(* CODESYS project tcprocess.library
   Company: TcNexa
   DefaultNamespace: TcNexa_Components_TcProcess
   Version: 1.0.0.0
   Placeholder: TcProcess
   Author: ATI Software Engineering
   Description: This library serves as a valuable resource for managing reusable components within your automation projects
   Title: TcProcess

Project tree, tasks and I/O mapping:
  libraries: Tc2_Standard, * (Beckhoff Automation GmbH); Tc2_System, * (Beckhoff Automation GmbH); Tc3_Module, * (Beckhoff Automation GmbH); TcUnit, * (www.tcunit.org)
  Process Method Response/
    function block FB_MethodResponse [ST]: _clear, busy, description, error, copyFrom, setBusy, setFail, setPass
    function block FB_MethodResponse_1 [ST]: _clear, _formatDescription, _formatErrorMsg, busy, description, error, errorId, errorMsg, errorSrc, statusId, statusMsg, copyFrom, setBusy, setFail, setPass
  Process Step/
    function block FB_ProcessStep [ST]: actual, FB_main, inc, init, onEntry, onExit, set
  Tests/
    function block FB_MethodResponse_Test [ST]: _t_01_SetResponsePass_ExpectResponsePass, _t_02_SetResponseFail_ExpectResponseFail, _t_03_SetResponseBusy_ExpectResponseBusy, _t_04_CopyFrom_ExpectSameResponse
    function block FB_ProcessStep_Test [ST]: _t_01_StepInc_ExpectStepInc, _t_02_StepSet100_ExpectStep100, _t_03_StepManagment
    program PRG_TEST [ST]
  Version/
    global variables Global_Version
*)

// Version/Global_Version
{attribute 'TcGenerated'}
{attribute 'no-analysis'}
{attribute 'linkalways'}
// This function has been automatically generated from the project information.
VAR_GLOBAL CONSTANT
	{attribute 'const_non_replaced'}
	stLibVersion_TcProcess : ST_LibVersion := (iMajor := 1, iMinor := 0, iBuild := 0, iRevision := 0, nFlags := 0, sVersion := '1.0.0.0');
END_VAR

// Process Method Response/FB_MethodResponse
FUNCTION_BLOCK FB_MethodResponse
VAR
	_busy			: BOOL;						// Indicates if the method call is in progress
	_error			: BOOL;						// Indicates if the method call failed
	_description	: Tc2_System.T_MaxString;	// Information to show to the user
	
	
	
	
//	_statusMsg		: Tc2_System.T_MaxString;	// Status message from method call
//	_statusId		: UDINT;					// Message ID from method call, for further processing (translation etc.)
//	_errorMsg		: Tc2_System.T_MaxString;	// Error message from method call
//	_errorId		: UDINT;					// Error ID from method call
//	_errorSrc		: STRING;					// Source for the error (Beckhoff, Keyence etc.)
END_VAR

METHOD PROTECTED _clear
VAR_INPUT
END_VAR
_busy:= FALSE;
_error:= FALSE;
_description:= '';
END_METHOD

PROPERTY PUBLIC busy : BOOL
GET
busy:= _busy;
END_GET
END_PROPERTY

PROPERTY PUBLIC description : Tc2_System.T_MaxString
GET
description:= _description;
END_GET
END_PROPERTY

PROPERTY PUBLIC error : BOOL
GET
error:= _error;
END_GET
END_PROPERTY

METHOD PUBLIC copyFrom
VAR_INPUT
	Response		: FB_MethodResponse;
END_VAR
_busy:= Response.busy;
_error:= Response.error;
_description:= Response.description;
END_METHOD

METHOD PUBLIC setBusy
VAR_INPUT
	description	 	: Tc2_System.T_MaxString;
END_VAR
_clear();

_busy:= TRUE;
_description:= description;
END_METHOD

METHOD PUBLIC setFail
VAR_INPUT
	description	 	: Tc2_System.T_MaxString;
END_VAR
_clear();

_error:= TRUE;
_description:= description;
END_METHOD

METHOD PUBLIC setPass
VAR_INPUT
END_VAR
_clear();
END_METHOD

END_FUNCTION_BLOCK

// Process Method Response/FB_MethodResponse_1
FUNCTION_BLOCK FB_MethodResponse_1
VAR
	_busy			: BOOL;						// Indicates if the method call is in progress
	_error			: BOOL;						// Indicates if the method call failed
	_description	: Tc2_System.T_MaxString;	// Status and error message combined from method call
	_statusMsg		: Tc2_System.T_MaxString;	// Status message from method call
	_statusId		: UDINT;					// Message ID from method call, for further processing (translation etc.)
	_errorMsg		: Tc2_System.T_MaxString;	// Error message from method call
	_errorId		: UDINT;					// Error ID from method call
	_errorSrc		: STRING;					// Source for the error (Beckhoff, Keyence etc.)
END_VAR

METHOD PROTECTED _clear
VAR_INPUT
END_VAR
_busy:= FALSE;
_error:= FALSE;
_description:= '';
_statusMsg:= '';
_statusId:= 0;
_errorMsg:= '';
_errorId:= 0;
_errorSrc:= '';
END_METHOD

METHOD PROTECTED _formatDescription
VAR_INPUT
END_VAR
IF (_statusMsg <> '') AND (_errorMsg <> '') THEN
	_description:= Tc2_Standard.CONCAT(
		STR1:= _statusMsg,
		STR2:= ' -> ');
	_description:= Tc2_Standard.CONCAT(
		STR1:= _description,
		STR2:= _errorMsg);
ELSIF (_statusMsg <> '') THEN
	_description:= _statusMsg;
ELSIF (_errorMsg <> '') THEN
	_description:= _errorMsg;
END_IF
END_METHOD

METHOD PROTECTED _formatErrorMsg
VAR_INPUT
	
END_VAR
IF (_errorMsg = '') THEN
	IF (_errorSrc <> '') AND (_errorId <> 0) THEN
		_errorMsg:= Tc2_Standard.CONCAT(
			STR1:= _errorSrc,
			STR2:= ' error code ');
		_errorMsg:= Tc2_Standard.CONCAT(
			STR1:= _errorMsg,
			STR2:= UDINT_TO_STRING(_errorId));
	ELSIF (_errorSrc <> '') THEN
		_errorMsg:= Tc2_Standard.CONCAT(
			STR1:= _errorSrc,
			STR2:= ' error');	
	ELSIF (_errorId <> 0) THEN
		_errorMsg:= Tc2_Standard.CONCAT(
			STR1:= 'Error code ',
			STR2:= UDINT_TO_STRING(_errorId));
	END_IF
END_IF
END_METHOD

PROPERTY PUBLIC busy : BOOL
GET
busy:= _busy;
END_GET
END_PROPERTY

PROPERTY PUBLIC description : Tc2_System.T_MaxString
GET
description:= _description;
END_GET
END_PROPERTY

PROPERTY PUBLIC error : BOOL
GET
error:= _error;
END_GET
END_PROPERTY

PROPERTY PUBLIC errorId : UDINT
GET
errorId:= _errorId;
END_GET
END_PROPERTY

PROPERTY PUBLIC errorMsg : Tc2_System.T_MaxString
GET
errorMsg:= _errorMsg;
END_GET
END_PROPERTY

PROPERTY PUBLIC errorSrc : STRING
GET
errorSrc:= _errorSrc;
END_GET
END_PROPERTY

PROPERTY PUBLIC statusId : UDINT
GET
statusId:= _statusId;
END_GET
END_PROPERTY

PROPERTY PUBLIC statusMsg : Tc2_System.T_MaxString
GET
statusMsg:= _statusMsg;
END_GET
END_PROPERTY

METHOD PUBLIC copyFrom
VAR_INPUT
	Response		: FB_MethodResponse_1;
END_VAR
_busy:= Response.busy;
_error:= Response.error;
_description:= Response.description;
_statusMsg:= Response.statusMsg;
_statusId:= Response.statusId;
_errorMsg:= Response.errorMsg;
_errorId:= Response.errorId;
_errorSrc:= Response.errorSrc;
END_METHOD

METHOD PUBLIC setBusy
VAR_INPUT
	statusMsg	 	: STRING;
	statusId		: UDINT;
END_VAR
_clear();

_busy:= TRUE;
_statusMsg:= statusMsg;
_statusId:= statusId;
_description:= statusMsg;
END_METHOD

METHOD PUBLIC setFail
VAR_INPUT
	statusMsg	 	: STRING;
	statusId		: UDINT;
	errorMsg	 	: STRING;
	errorId			: UDINT;
	errorSrc	 	: STRING;
END_VAR
_clear();

_error:= TRUE;
_statusMsg:= statusMsg;
_statusId:= statusId;
_errorMsg:= errorMsg;
_errorId:= errorId;
_errorSrc:= errorSrc;

_formatErrorMsg();
_formatDescription();
END_METHOD

METHOD PUBLIC setPass
VAR_INPUT
END_VAR
_clear();
END_METHOD

END_FUNCTION_BLOCK

// Process Step/FB_ProcessStep
FUNCTION_BLOCK FB_ProcessStep
VAR
	_actual						: INT:= -1;
	_target						: INT;
	_onEntry					: BOOL;
	_onExit						: BOOL;
END_VAR

PROPERTY PUBLIC actual : INT
GET
PUBLIC 
VAR
END_VAR
actual:= _actual;
END_GET
END_PROPERTY

METHOD PUBLIC FB_main
VAR_INPUT
END_VAR
_onEntry:= _actual <> _target;
_actual:= _target;

_onExit:= FALSE;
END_METHOD

METHOD PUBLIC inc : FB_MethodResponse
VAR
END_VAR
IF (_actual + 1) < _actual THEN
	inc.setFail(description:= 'Overflow _actual');
ELSE
	_target:= _actual + 1;
	_onExit:= TRUE;
	inc.setPass();
END_IF
END_METHOD

METHOD PUBLIC init
VAR_INPUT
END_VAR
_target:= 0;
_onEntry:= FALSE;
_onExit:= FALSE;
END_METHOD

PROPERTY PUBLIC onEntry : BOOL
GET
onEntry:= _onEntry;
END_GET
END_PROPERTY

PROPERTY PUBLIC onExit : BOOL
GET
onExit:= _onExit;
END_GET
END_PROPERTY

METHOD PUBLIC set : FB_MethodResponse
VAR_INPUT
	target	: INT;
END_VAR
IF (target < 0) THEN
	set.setFail(description:= 'Invalid target (< 0)');
ELSE
	_target:= target;
	_onExit:= TRUE;	
	set.setPass();
END_IF
END_METHOD

END_FUNCTION_BLOCK

// Tests/FB_MethodResponse_Test
FUNCTION_BLOCK INTERNAL FB_MethodResponse_Test EXTENDS TcUnit.FB_TestSuite
VAR_INPUT
END_VAR
VAR_OUTPUT
END_VAR
VAR
END_VAR

_t_01_SetResponsePass_ExpectResponsePass();
_t_02_SetResponseFail_ExpectResponseFail();
_t_03_SetResponseBusy_ExpectResponseBusy();
_t_04_CopyFrom_ExpectSameResponse();

METHOD PROTECTED _t_01_SetResponsePass_ExpectResponsePass
VAR
	_MethodResponse			: FB_MethodResponse_1;
END_VAR
TcUnit.TEST('_t_01_SetResponsePass_ExpectResponsePass');

_MethodResponse.setPass();	

AssertEquals_STRING	(Expected:= '',
					Actual:= _MethodResponse.statusMsg,
					Message:= 'message missmatch');

AssertEquals_UDINT	(Expected:= 0,
					Actual:= _MethodResponse.statusId,
					Message:= 'messageId missmatch');

AssertEquals_STRING	(Expected:= '',
					Actual:= _MethodResponse.errorMsg,
					Message:= 'errorMsg missmatch');

AssertEquals_UDINT	(Expected:= 0,
					Actual:= _MethodResponse.errorId,
					Message:= 'errorId missmatch');

AssertEquals_STRING	(Expected:= '',
					Actual:= _MethodResponse.errorSrc,
					Message:= 'errorSrc missmatch');

AssertEquals_STRING	(Expected:= '',
					Actual:= _MethodResponse.description,
					Message:= 'description missmatch');
					
AssertFalse			(Condition:= _MethodResponse.error,
					Message:= 'error is not FALSE');		
					
AssertFalse			(Condition:= _MethodResponse.busy,
					Message:= 'busy is not FALSE');			

TcUnit.TEST_FINISHED();
END_METHOD

METHOD PROTECTED _t_02_SetResponseFail_ExpectResponseFail
VAR
	_MethodResponse			: FB_MethodResponse_1;
END_VAR
TcUnit.TEST('_t_02_SetResponseFail_ExpectResponseFail');

(* Fail without statusMsg & errorMsg & errorSrc *)
_MethodResponse.setFail(
	statusMsg:= '',
	statusId:= 2,
	errorMsg:= '',
	errorId:= 0,
	errorSrc:= '');

AssertEquals_STRING	(Expected:= '',
					Actual:= _MethodResponse.statusMsg,
					Message:= 'message missmatch');

AssertEquals_UDINT	(Expected:= 2,
					Actual:= _MethodResponse.statusId,
					Message:= 'messageId missmatch');

AssertEquals_STRING	(Expected:= '',
					Actual:= _MethodResponse.errorMsg,
					Message:= 'errorMsg missmatch');

AssertEquals_UDINT	(Expected:= 0,
					Actual:= _MethodResponse.errorId,
					Message:= 'errorId missmatch');

AssertEquals_STRING	(Expected:= '',
					Actual:= _MethodResponse.errorSrc,
					Message:= 'errorSrc missmatch');

AssertEquals_STRING	(Expected:= '',
					Actual:= _MethodResponse.description,
					Message:= 'description missmatch');
					
AssertTrue			(Condition:= _MethodResponse.error,
					Message:= 'error is not TRUE');		
					
AssertFalse			(Condition:= _MethodResponse.busy,
					Message:= 'busy is not FALSE');	

(* Fail without errorMsg & errorSrc *)
_MethodResponse.setFail(
	statusMsg:= 'Fail description',
	statusId:= 3,
	errorMsg:= '',
	errorId:= 0,
	errorSrc:= '');

AssertEquals_STRING	(Expected:= 'Fail description',
					Actual:= _MethodResponse.statusMsg,
					Message:= 'message missmatch');

AssertEquals_UDINT	(Expected:= 3,
					Actual:= _MethodResponse.statusId,
					Message:= 'messageId missmatch');

AssertEquals_STRING	(Expected:= '',
					Actual:= _MethodResponse.errorMsg,
					Message:= 'errorMsg missmatch');

AssertEquals_UDINT	(Expected:= 0,
					Actual:= _MethodResponse.errorId,
					Message:= 'errorId missmatch');

AssertEquals_STRING	(Expected:= '',
					Actual:= _MethodResponse.errorSrc,
					Message:= 'errorSource missmatch');

AssertEquals_STRING	(Expected:= 'Fail description',
					Actual:= _MethodResponse.description,
					Message:= 'description missmatch');
					
AssertTrue			(Condition:= _MethodResponse.error,
					Message:= 'error is not TRUE');		
					
AssertFalse			(Condition:= _MethodResponse.busy,
					Message:= 'busy is not FALSE');	
					
(* Fail without errorSrc *)
_MethodResponse.setFail(
	statusMsg:= 'Fail description',
	statusId:= 3,
	errorMsg:= 'Error description',
	errorId:= 4,
	errorSrc:= '');

AssertEquals_STRING	(Expected:= 'Fail description',
					Actual:= _MethodResponse.statusMsg,
					Message:= 'message missmatch');

AssertEquals_UDINT	(Expected:= 3,
					Actual:= _MethodResponse.statusId,
					Message:= 'messageId missmatch');

AssertEquals_STRING	(Expected:= 'Error description',
					Actual:= _MethodResponse.errorMsg,
					Message:= 'errorMsg missmatch');

AssertEquals_UDINT	(Expected:= 4,
					Actual:= _MethodResponse.errorId,
					Message:= 'errorId missmatch');

AssertEquals_STRING	(Expected:= '',
					Actual:= _MethodResponse.errorSrc,
					Message:= 'errorSource missmatch');

AssertEquals_STRING	(Expected:= 'Fail description -> Error description',
					Actual:= _MethodResponse.description,
					Message:= 'description missmatch');
					
AssertTrue			(Condition:= _MethodResponse.error,
					Message:= 'error is not TRUE');		
					
AssertFalse			(Condition:= _MethodResponse.busy,
					Message:= 'busy is not FALSE');		
					
(* Fail without statusMsg & errorSrc *)
_MethodResponse.setFail(
	statusMsg:= '',
	statusId:= 5,
	errorMsg:= 'Error description',
	errorId:= 4,
	errorSrc:= '');

AssertEquals_STRING	(Expected:= '',
					Actual:= _MethodResponse.statusMsg,
					Message:= 'message missmatch');

AssertEquals_UDINT	(Expected:= 5,
					Actual:= _MethodResponse.statusId,
					Message:= 'messageId missmatch');

AssertEquals_STRING	(Expected:= 'Error description',
					Actual:= _MethodResponse.errorMsg,
					Message:= 'errorMsg missmatch');

AssertEquals_UDINT	(Expected:= 4,
					Actual:= _MethodResponse.errorId,
					Message:= 'errorId missmatch');

AssertEquals_STRING	(Expected:= '',
					Actual:= _MethodResponse.errorSrc,
					Message:= 'errorSource missmatch');

AssertEquals_STRING	(Expected:= 'Error description',
					Actual:= _MethodResponse.description,
					Message:= 'description missmatch');
					
AssertTrue			(Condition:= _MethodResponse.error,
					Message:= 'error is not TRUE');		
					
AssertFalse			(Condition:= _MethodResponse.busy,
					Message:= 'busy is not FALSE');	
					
(* Fail *)
_MethodResponse.setFail(
	statusMsg:= 'Fail description',
	statusId:= 3,
	errorMsg:= 'Error description',
	errorId:= 4,
	errorSrc:= 'Beckhoff');

AssertEquals_STRING	(Expected:= 'Fail description',
					Actual:= _MethodResponse.statusMsg,
					Message:= 'message missmatch');

AssertEquals_UDINT	(Expected:= 3,
					Actual:= _MethodResponse.statusId,
					Message:= 'messageId missmatch');

AssertEquals_STRING	(Expected:= 'Error description',
					Actual:= _MethodResponse.errorMsg,
					Message:= 'errorMsg missmatch');

AssertEquals_UDINT	(Expected:= 4,
					Actual:= _MethodResponse.errorId,
					Message:= 'errorId missmatch');

AssertEquals_STRING	(Expected:= 'Beckhoff',
					Actual:= _MethodResponse.errorSrc,
					Message:= 'errorSource missmatch');

AssertEquals_STRING	(Expected:= 'Fail description -> Error description',
					Actual:= _MethodResponse.description,
					Message:= 'description missmatch');
					
AssertTrue			(Condition:= _MethodResponse.error,
					Message:= 'error is not TRUE');		
					
AssertFalse			(Condition:= _MethodResponse.busy,
					Message:= 'busy is not FALSE');	
					
(* Fail without errorMsg *)
_MethodResponse.setFail(
	statusMsg:= 'Fail description',
	statusId:= 3,
	errorMsg:= '',
	errorId:= 4,
	errorSrc:= 'Beckhoff');

AssertEquals_STRING	(Expected:= 'Fail description',
					Actual:= _MethodResponse.statusMsg,
					Message:= 'message missmatch');

AssertEquals_UDINT	(Expected:= 3,
					Actual:= _MethodResponse.statusId,
					Message:= 'messageId missmatch');

AssertEquals_STRING	(Expected:= 'Beckhoff error code 4',
					Actual:= _MethodResponse.errorMsg,
					Message:= 'errorMsg missmatch');

AssertEquals_UDINT	(Expected:= 4,
					Actual:= _MethodResponse.errorId,
					Message:= 'errorId missmatch');

AssertEquals_STRING	(Expected:= 'Beckhoff',
					Actual:= _MethodResponse.errorSrc,
					Message:= 'errorSource missmatch');

AssertEquals_STRING	(Expected:= 'Fail description -> Beckhoff error code 4',
					Actual:= _MethodResponse.description,
					Message:= 'description missmatch');
					
AssertTrue			(Condition:= _MethodResponse.error,
					Message:= 'error is not TRUE');		
					
AssertFalse			(Condition:= _MethodResponse.busy,
					Message:= 'busy is not FALSE');		

TcUnit.TEST_FINISHED();
END_METHOD

METHOD PROTECTED _t_03_SetResponseBusy_ExpectResponseBusy
VAR
	_MethodResponse			: FB_MethodResponse_1;
END_VAR
TcUnit.TEST('_t_03_SetResponseBusy_ExpectResponseBusy');

_MethodResponse.setBusy(
	statusMsg:= 'Busy description', 
	statusId:= 3);

AssertEquals_STRING	(Expected:= 'Busy description',
					Actual:= _MethodResponse.statusMsg,
					Message:= 'message missmatch');

AssertEquals_UDINT	(Expected:= 3,
					Actual:= _MethodResponse.statusId,
					Message:= 'messageId missmatch');

AssertEquals_STRING	(Expected:= '',
					Actual:= _MethodResponse.errorMsg,
					Message:= 'errorMsg missmatch');

AssertEquals_UDINT	(Expected:= 0,
					Actual:= _MethodResponse.errorId,
					Message:= 'errorId missmatch');

AssertEquals_STRING	(Expected:= '',
					Actual:= _MethodResponse.errorSrc,
					Message:= 'errorSrc missmatch');

AssertEquals_STRING	(Expected:= 'Busy description',
					Actual:= _MethodResponse.description,
					Message:= 'description missmatch');
					
AssertFalse			(Condition:= _MethodResponse.error,
					Message:= 'error is not FALSE');		
					
AssertTrue			(Condition:= _MethodResponse.busy,
					Message:= 'busy is not TRUE');		

TcUnit.TEST_FINISHED();
END_METHOD

METHOD PROTECTED _t_04_CopyFrom_ExpectSameResponse
VAR
	_ControlResponse		: FB_MethodResponse_1;
	_MethodResponse			: FB_MethodResponse_1;
END_VAR
TcUnit.TEST('_t_04_CopyFrom_ExpectSameResponse');

_ControlResponse.setFail(
	statusMsg:= 'Fail description',
	statusId:= 3,
	errorMsg:= 'Error description',
	errorId:= 4,
	errorSrc:= 'Beckhoff');
_MethodResponse.copyFrom(Response:= _ControlResponse);

AssertEquals_STRING	(Expected:= 'Fail description',
					Actual:= _MethodResponse.statusMsg,
					Message:= 'message missmatch');

AssertEquals_UDINT	(Expected:= 3,
					Actual:= _MethodResponse.statusId,
					Message:= 'messageId missmatch');

AssertEquals_STRING	(Expected:= 'Error description',
					Actual:= _MethodResponse.errorMsg,
					Message:= 'errorMsg missmatch');

AssertEquals_UDINT	(Expected:= 4,
					Actual:= _MethodResponse.errorId,
					Message:= 'errorId missmatch');

AssertEquals_STRING	(Expected:= 'Beckhoff',
					Actual:= _MethodResponse.errorSrc,
					Message:= 'errorSource missmatch');

AssertEquals_STRING	(Expected:= 'Fail description -> Error description',
					Actual:= _MethodResponse.description,
					Message:= 'description missmatch');
					
AssertTrue			(Condition:= _MethodResponse.error,
					Message:= 'error is not TRUE');		
					
AssertFalse			(Condition:= _MethodResponse.busy,
					Message:= 'busy is not FALSE');			

TcUnit.TEST_FINISHED();
END_METHOD

END_FUNCTION_BLOCK

// Tests/FB_ProcessStep_Test
FUNCTION_BLOCK INTERNAL FB_ProcessStep_Test EXTENDS TcUnit.FB_TestSuite
VAR
END_VAR

_t_01_StepInc_ExpectStepInc();
_t_02_StepSet100_ExpectStep100();
_t_03_StepManagment();

METHOD PRIVATE _t_01_StepInc_ExpectStepInc
VAR
	_Step 		: FB_ProcessStep;
END_VAR
TcUnit.TEST('_t_01_StepInc_ExpectStepInc');

_Step.init();
_Step.FB_main();
_Step.FB_main();	// simulate 2 cycles
(* PLC Cycle 1*)
_Step.inc();

AssertFalse			(Condition:= _Step.onEntry,
					Message:= 'onEntry is not FALSE');
            		
AssertTrue			(Condition:= _Step.onExit,
					Message:= 'onExit is not TRUE');
			
AssertEquals_INT	(Expected:= 0,
					Actual:= _Step.actual,
					Message:= 'actual is not 0');
(* PLC Cycle 2*)
_Step.FB_main();

AssertTrue			(Condition:= _Step.onEntry,
					Message:= 'onEntry is not TRUE');
            		
AssertFalse			(Condition:= _Step.onExit,
					Message:= 'onExit is not FALSE');
			
AssertEquals_INT	(Expected:= 1,
					Actual:= _Step.actual,
					Message:= 'actual is not 1');

TcUnit.TEST_FINISHED();
END_METHOD

METHOD PRIVATE _t_02_StepSet100_ExpectStep100
VAR
	_Step 		: FB_ProcessStep;
END_VAR
TcUnit.TEST('_t_02_StepSet100_ExpectStep100');

_Step.init();
_Step.FB_main();
_Step.FB_main();	// simulate 2 cycles
(* PLC Cycle 1*)
_Step.set(target:= 100);

AssertFalse			(Condition:= _Step.onEntry,
					Message:= 'onEntry is not FALSE');
            		
AssertTrue			(Condition:= _Step.onExit,
					Message:= 'onExit is not TRUE');
			
AssertEquals_INT	(Expected:= 0,
					Actual:= _Step.actual,
					Message:= 'actual is not 0');
(* PLC Cycle 2*)
_Step.FB_main();

AssertTrue			(Condition:= _Step.onEntry,
					Message:= 'onEntry is not TRUE');
            		
AssertFalse			(Condition:= _Step.onExit,
					Message:= 'onExit is not FALSE');
			
AssertEquals_INT	(Expected:= 100,
					Actual:= _Step.actual,
					Message:= 'actual is not 100');

TcUnit.TEST_FINISHED();
END_METHOD

METHOD PRIVATE _t_03_StepManagment
VAR_INST
	_Step 					: FB_ProcessStep;
	_Step1_Timer			: Tc2_Standard.TON;
	_Step2_Timer			: Tc2_Standard.TON;
	_init					: BOOL;
	_i 						: INT:= 0;
	_stepOnEntryCounter		: INT;
	_stepOnExitCounter		: INT;
END_VAR
TcUnit.TEST('_t_03_StepManagment');

IF NOT _init THEN
	_Step.init();
	_init:= TRUE;
END_IF

_Step1_Timer(IN:= (_Step.actual = 1), PT:= T#100MS);
_Step2_Timer(IN:= (_Step.actual = 2), PT:= T#500MS);
_Step.FB_main();

CASE _Step.actual OF
0:
	IF _Step.onEntry THEN
		_stepOnEntryCounter:= _stepOnEntryCounter + 1;
	END_IF
	
	_Step.inc();
	
	IF _Step.onExit THEN
		_stepOnExitCounter:= _stepOnExitCounter + 1;
	END_IF
1:
	IF _Step.onEntry THEN
		_stepOnEntryCounter:= _stepOnEntryCounter + 1;
	END_IF
	
	IF _Step1_Timer.Q THEN
		_Step.set(2);
	END_IF
	
	IF _Step.onExit THEN
		_stepOnExitCounter:= _stepOnExitCounter + 1;
	END_IF
2:
	IF _Step.onEntry THEN
		_stepOnEntryCounter:= _stepOnEntryCounter + 1;
	END_IF
	
	IF _Step2_Timer.Q THEN
		_Step.inc();		
	END_IF
	
	IF _Step.onExit THEN
		_stepOnExitCounter:= _stepOnExitCounter + 1;
	END_IF
3:
	AssertEquals_INT(Expected:= 3,
					Actual:= _stepOnEntryCounter,
					Message:= '_stepOnEntryCounter is not 3');
	AssertEquals_INT(Expected:= 3,
					Actual:= _stepOnExitCounter,
					Message:= '_stepOnExitCounter is not 3');

	TcUnit.TEST_FINISHED();
END_CASE
END_METHOD

END_FUNCTION_BLOCK

// Tests/PRG_TEST
PROGRAM PRG_TEST
VAR
	_Step_Test				: FB_ProcessStep_Test;
	_MethodResp_Test		: FB_MethodResponse_Test;
END_VAR

TcUnit.RUN();

END_PROGRAM
